// TIA Portal V20 export
TYPE "LER_typeBrakeTestUnitCommands"
// stored: Access Published
   STRUCT
      allStart : Bool;
      allStop : Bool;
   END_STRUCT;
END_TYPE
